// TwinCAT 3 PLC project FileWritingStateMachine
// ProgramVersion: 3.1.4024.0
// libraries:
//   Tc2_Standard, * (Beckhoff Automation GmbH)
//   Tc2_System, * (Beckhoff Automation GmbH)
//   Tc3_Module, * (Beckhoff Automation GmbH)
// project tree:
//   DUTs/ ST_Event.TcDUT
//   / PlcTask.TcTTO
//   POUs/ FB_CsvFileWriter.TcPOU, I_FileWriter.TcIO, MAIN.TcPOU
// (motion and I/O tree: see PLC project instructions_practice)
// real-time tasks:
//   TASK PlcTask: cycle T#10ms, priority 20, ADS port 350
//   TASK PlcTask1: cycle T#10ms, priority 22, ADS port 351
//   TASK PlcTask2: cycle T#10ms, priority 21, ADS port 352

CONFIGURATION FileWritingStateMachine
    RESOURCE PLC ON TwinCAT3
        TASK PlcTask(INTERVAL := T#10ms, PRIORITY := 21);
        PROGRAM MAIN WITH PlcTask : MAIN;
    END_RESOURCE
END_CONFIGURATION

// ---- DUTs/ST_Event.TcDUT
TYPE ST_Event :
STRUCT
	

END_STRUCT
END_TYPE

// ---- POUs/I_FileWriter.TcIO
INTERFACE I_FileWriter

METHOD WriteEvent : BOOL
VAR_INPUT
	sMessage : STRING ;
END_VAR
END_METHOD

END_INTERFACE

// ---- POUs/MAIN.TcPOU
PROGRAM MAIN
VAR
	bStart : BOOL;
	fbCsv : FB_CsvFileWriter;
	iFileWriter : I_FileWriter;
	sMessage : STRING := 'This is third message in the file';
END_VAR

iFileWriter := fbCsv;

IF bStart THEN
	iFileWriter.WriteEvent(sMessage);
	bStart := FALSE;
END_IF
fbCsv();

END_PROGRAM

// ---- POUs/FB_CsvFileWriter.TcPOU
FUNCTION_BLOCK FB_CsvFileWriter IMPLEMENTS I_FileWriter

VAR
	sMessageString : STRING;
	eWriteState : (FILE_OPEN_TRIGGER, FILE_OPEN, WAIT_FOR_EVENT, WRITE_EVENT_TRIGGER, WRITE_EVENT,FILE_CLOSE_TRIGGER, FILE_CLOSE, ERROR );
	fbFileOpen : FB_FileOpen := (sPathName := 'C:\Users\kameshwaran.k\OneDrive - InTimeTec Visionsoft Pvt. Ltd.,\Documents/Event.txt', nMode := FOPEN_MODEAPPEND OR FOPEN_MODETEXT);
	fbFilePuts : FB_FilePuts;
	fbFileClose : FB_FileClose;
	sCsvString : T_MaxString ;
END_VAR

CASE eWriteState OF
	FILE_OPEN_TRIGGER:
	fbFileOpen(bExecute := TRUE);
	eWriteState := FILE_OPEN;
	
	FILE_OPEN:
	fbFileOpen(bExecute := FALSE);
	IF fbFileOpen.bError THEN
		eWriteState := ERROR;
		ELSIF NOT fbFileOpen.bBusy AND fbFileOpen.hFile <> 0 THEN
			eWriteState := WAIT_FOR_EVENT;
	END_IF
	WAIT_FOR_EVENT:	
	//No logic 
	
	WRITE_EVENT_TRIGGER:
	sCsvString := ConvertString(sString := sMessageString);
	fbFilePuts(bExecute := TRUE, sLine := sCsvString, hFile := fbFileOpen.hFile);
	eWriteState := WRITE_EVENT;
	
	WRITE_EVENT:
	fbFilePuts(bExecute := FALSE);
	IF fbFilePuts.bError THEN
		eWriteState := ERROR;
		ELSIF NOT fbFilePuts.bBusy THEN
			eWriteState := FILE_CLOSE_TRIGGER;
			
	END_IF
	
	FILE_CLOSE_TRIGGER:
	fbFileClose(bExecute := TRUE, hFile := fbFileOpen.hFile);
	eWriteState := FILE_CLOSE;
	
	FILE_CLOSE:
	fbFileClose(bExecute := FALSE);
	IF fbFileClose.bError THEN
		eWriteState := ERROR;
		ELSIF NOT fbFileClose.bBusy THEN
			eWriteState := FILE_OPEN_TRIGGER;
	END_IF
	ERROR:
END_CASE

METHOD PRIVATE ConvertString : T_MaxString
VAR_INPUT
	sString : STRING;
END_VAR
ConvertString := CONCAT(STR1 := sString , STR2 := '$n');
END_METHOD

{warning 'add method implementation '}
METHOD WriteEvent : BOOL
VAR_INPUT
	sMessage : STRING ;
END_VAR
IF eWriteState = WAIT_FOR_EVENT THEN
	eWriteState := WRITE_EVENT_TRIGGER;
	sMessageString := sMessage;
END_IF
END_METHOD

END_FUNCTION_BLOCK
